Fanuc KAREL source: kt00537.KL

PROGRAM KT00537
%STACKSIZE=65535
%PRIORITY=65535
%NOLOCKGROUP
VAR
P1 : JOINTPOS9
P2 : POSITION
OUT : JOINTPOS9
BEGIN
-- UNRESOLVED_PC line 8 opcodes [49 7E 49 60 7E 4A] marker_code=0
END KT00537
